(* Schneider Machine Expert - Basic project 5 Run-2 Stop (1T), file version 2.7.0.0 *)
(* ProjectInformations: Name=New project *)

HARDWARE
  Cpu 0: TM200C32R
  EthernetConfiguration: NetworkName=M200, IpAllocationMode=FixedAddress, IpAddress=0.0.0.0, SubnetMask=0.0.0.0
  SerialLineConfiguration: Baud=Baud19200, Parity=ParityEven, DataBits=DataBits8, StopBits=StopBits1, PhysicalMedium=PhysicalMediumRs485, TransmissionMode=TransmissionModeModbusRtu, SlaveId=1, Addressing=SlaveAddressing
  MastTask: UsePeriodScanMode=false, PeriodScan=100
  FastTask: Period=255
  CpuBehavior: StartingMode=StartAsPreviousState, AutoSaveRamOnEeprom=true, WatchdogPeriod=250

SYMBOLS  (address, symbol, comment, settings)
  %M0         "X"
  %M1         "T1 DN"
  %M2         "C1 DN"
  %M3         "C2 DN"
  %TM0        [Preset=1000, Base=OneMilliSeconds]
  %C1         [Preset=5]
  %C2         [Preset=10]
  %I0.0       "START"
  %I0.1       "STOP"
  %Q0.0       "Motor"

POU New POU
  (* SectionNumber=1 *)

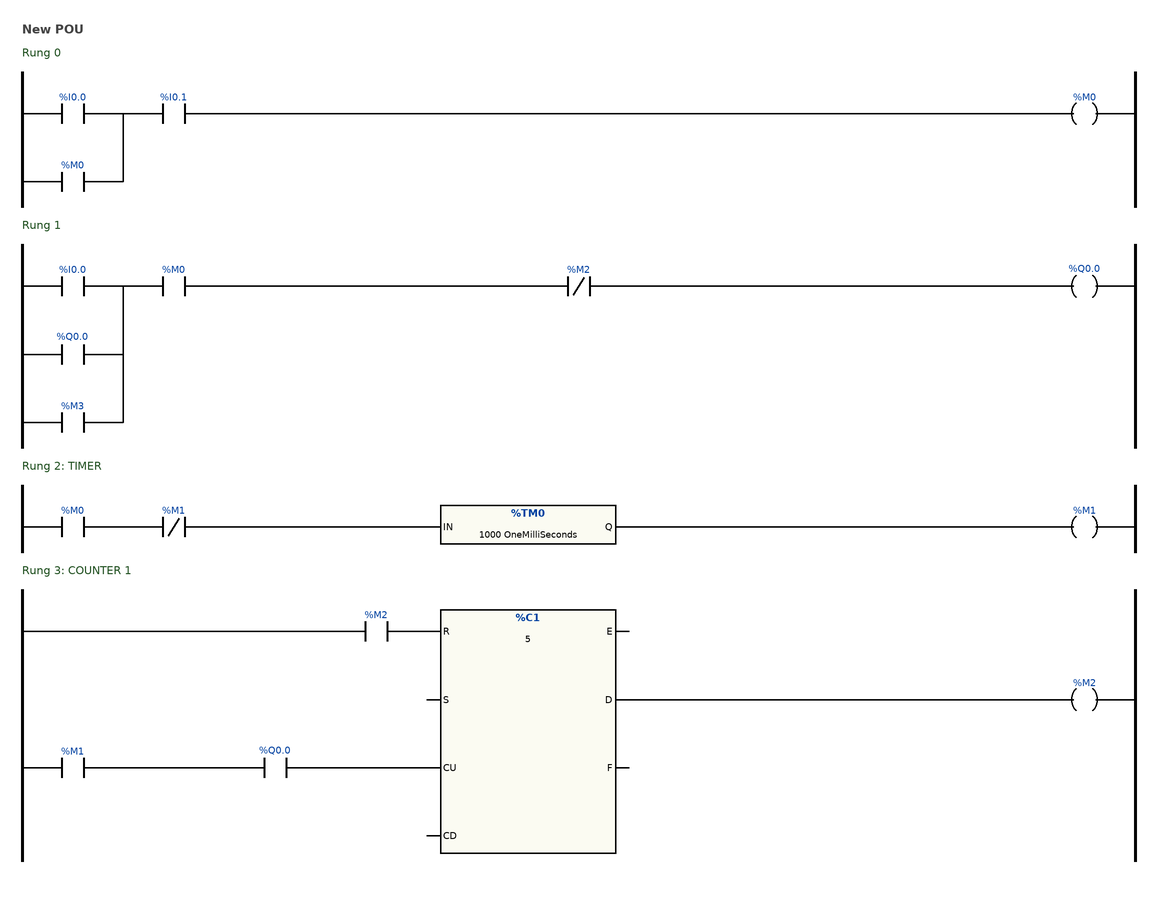

// Rung 0
  LD %I0.0
  OR %M0
  AND %I0.1
  ST %M0
  // as ST:
  //   %M0 := (%I0.0 OR %M0) AND %I0.1;

// Rung 1
  LD %I0.0
  OR %Q0.0
  OR %M3
  AND %M0
  ANDN %M2
  ST %Q0.0
  // as ST:
  //   %Q0.0 := (%I0.0 OR %Q0.0 OR %M3) AND %M0 AND NOT %M2;

// Rung 2: TIMER
  BLK %TM0
  LD %M0
  ANDN %M1
  IN
  OUT_BLK
  LD Q
  ST %M1
  END_BLK
  // as ST:
  //   %TM0(IN := %M0 AND NOT %M1);
  //   %M1 := %TM0.Q;

// Rung 3: COUNTER 1
  BLK %C1
  LD %M2
  R
  LD %M1
  AND %Q0.0
  CU
  OUT_BLK
  LD D
  ST %M2
  END_BLK
  // as ST:
  //   %C1(R := %M2, CU := %M1 AND %Q0.0);
  //   %M2 := %C1.D;

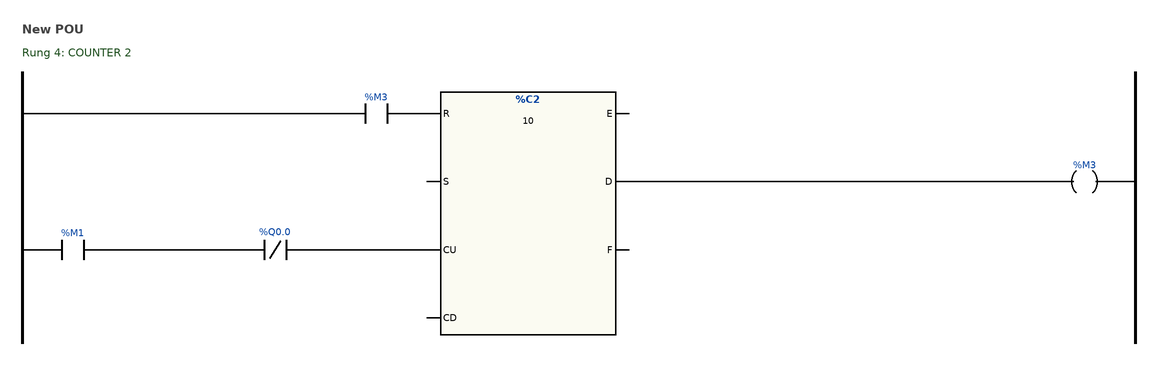

// Rung 4: COUNTER 2
  BLK %C2
  LD %M3
  R
  LD %M1
  ANDN %Q0.0
  CU
  OUT_BLK
  LD D
  ST %M3
  END_BLK
  // as ST:
  //   %C2(R := %M3, CU := %M1 AND NOT %Q0.0);
  //   %M3 := %C2.D;
